SUBAPPLICATION Ventilsteuerung_Uebung_011 (* Numeric Value Input *)
  (* Standard: 61499-2 *)
  (* Version 1.0, 2023-10-23, franz *)
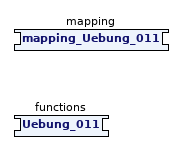
  SUBAPPS
    mapping : mapping_Uebung_011;
    functions : Uebung_011;
  END_SUBAPPS
END_SUBAPPLICATION
